Universal Robots PolyScope program: cottonMake.urp

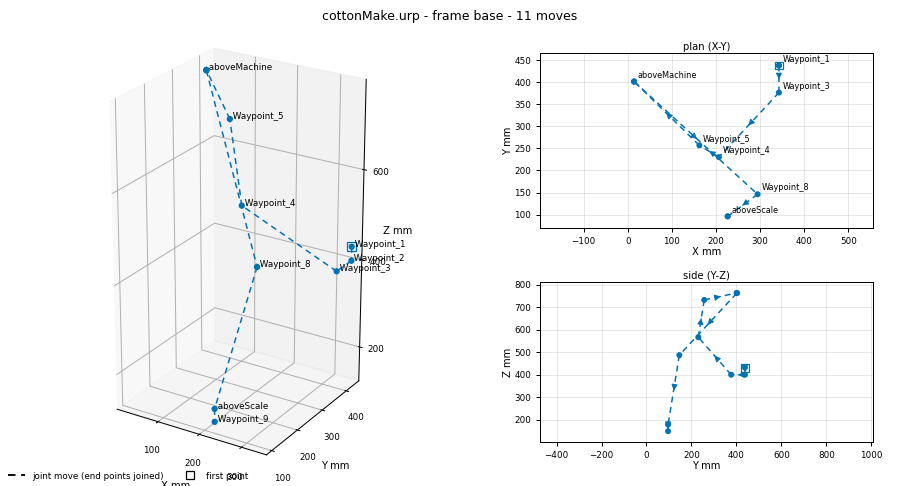
[picture p0: tool path of cottonMake.urp in frame base, 11 of 18 moves have a stored position in this frame; points joined in program order, loops and branches not executed]
Program cottonMake (installation=default directory=/programs/DavidMelin createdIn=5.12.4.1101661 lastSavedIn=5.12.4.1101661 robotSerialNumber=20225502378)
Calibrated DH parameters: a=[0.00022, -0.425328, -0.389701, 0.000059, 0.000065, 0]; d=[0.162608, 0.803456, 9.992211, -10.662202, 0.099702, 0.099559]; alpha=[1.570756, 0.001543, 0.004316, 1.570651, -1.570122, 0]; deltaTheta=[0, 0.002917, 0.116094, -0.119008, 0, -0.000001]
Robot Program (runOnlyOnce=true)
  circCenter := p[0.07107,0.64512,0.54131,0,2.2222,2.2222]
  radius := 0.12
  cBot := pose_add(circCenter, p[0,-radius,0,0,0,0])
  cLeft := pose_add(circCenter, p[-radius,0,0,0,0,0])
  cTop := pose_add(circCenter, p[0,radius,0,0,0,0])
  cRight := pose_add(circCenter, p[radius,0,0,0,0,0])
  Loops := 3
  URCap Gripper (Robotiq_Grippers, Robotiq Inc.) dataModel(position=0.0, force=0.0, speed=0.0, positionInDouble=0.0, forceInDouble=0.0, speedInDouble=0.0, slaveIds=[9], blocking=true)
  MoveJ speed 60 deg/s, acceleration 80 deg/s^2 (useActiveTCP=true) feature=Base
    Waypoint Waypoint (Variable): variable=cotonHomePos
    Waypoint Waypoint_1: TCP in base x=342.664 y=437.884 z=432.107 mm, rx=3.1413 ry=-0.0387 rz=0 rad; joints [65.941, -96.893, -90.985, -82.164, 90.259, -22.738] deg
    Waypoint Waypoint_2: TCP in base x=342.659 y=437.882 z=400.544 mm, rx=3.1413 ry=-0.0387 rz=0 rad; joints [65.938, -97.638, -94.818, -77.583, 90.259, -22.722] deg
  URCap Gripper (Robotiq_Grippers, Robotiq Inc.) dataModel(position=100.0, force=0.0, speed=0.0, positionInDouble=100.0, forceInDouble=0.0, speedInDouble=0.0, slaveIds=[9], blocking=true)
  MoveJ speed 60 deg/s, acceleration 80 deg/s^2 (useActiveTCP=true) feature=Base
    Waypoint Waypoint_3: TCP in base x=342.674 y=376.601 z=400.529 mm, rx=3.1413 ry=-0.0388 rz=0 rad; joints [62.998, -91.205, -101.8, -77.036, 90.249, -25.658] deg
    Waypoint Waypoint_4: TCP in base x=206.614 y=230.365 z=567.394 mm, rx=-2.941 ry=-0.1771 rz=0.13 rad; joints [70.752, -61.526, -101.667, -98.574, 99.079, -25.658] deg
    Waypoint Waypoint_5: TCP in base x=162.312 y=256.881 z=733.059 mm, rx=1.0793 ry=1.2981 rz=1.5955 rad; joints [107.929, -56.169, -91.557, -124.534, -6.229, -80.259] deg
    Waypoint aboveMachine: TCP in base x=14.31 y=401.62 z=764.278 mm, rx=-0.0463 ry=2.2239 rz=2.2128 rad; joints [113.283, -89.095, -46.167, -225.083, -68.031, -1.075] deg
  Loop While (checkContinuously=false) expression=Loops>0
    MoveP speed 250 mm/s, acceleration 1200 mm/s^2 (blendRadius=0.125 useActiveTCP=true) feature=Base
      Waypoint Waypoint (Variable): variable=cBot
      CircleMove (OrientationMode=UNCONSTRAINED)
        Waypoint Waypoint (Variable): variable=cRight
        Waypoint Waypoint (Variable): variable=cTop
    MoveP speed 250 mm/s, acceleration 1200 mm/s^2 (blendRadius=0.025 useActiveTCP=true) feature=Base
      Waypoint Waypoint (Variable): variable=cTop
      CircleMove (OrientationMode=UNCONSTRAINED)
        Waypoint Waypoint (Variable): variable=cLeft
        Waypoint Waypoint (Variable): variable=cBot
    Loops := Loops - 1
  MoveJ speed 60 deg/s, acceleration 80 deg/s^2 (useActiveTCP=true) feature=Base
    Waypoint aboveMachine: TCP in base x=14.31 y=401.62 z=764.278 mm, rx=-0.0463 ry=2.2239 rz=2.2128 rad; joints [113.283, -89.095, -46.167, -225.083, -68.031, -1.075] deg
    Waypoint Waypoint_6: TCP in base x=14.523 y=401.528 z=763.071 mm, rx=-1.5836 ry=0.0041 rz=0.0315 rad; joints [113.257, -89.129, -46.231, -225.448, -68.036, 181.754] deg
    Waypoint Waypoint_8: TCP in base x=294.267 y=146.163 z=487.658 mm, rx=-1.6041 ry=-0.2565 rz=0.2618 rad; joints [33.077, -80.074, -98.689, -191.144, -165.647, 171.099] deg
    Waypoint aboveScale: TCP in base x=226.497 y=96.066 z=178.622 mm, rx=-1.5818 ry=-0.3301 rz=0.3435 rad; joints [31.277, -91.949, -140.091, -142.239, -172.906, 166.771] deg
    Waypoint Waypoint_9: TCP in base x=226.483 y=96.053 z=149.343 mm, rx=-1.5818 ry=-0.3301 rz=0.3435 rad; joints [31.27, -97.11, -141.687, -135.565, -172.89, 166.689] deg
  URCap Gripper (Robotiq_Grippers, Robotiq Inc.) dataModel(position=0.0, force=0.0, speed=0.0, positionInDouble=0.0, forceInDouble=0.0, speedInDouble=0.0, slaveIds=[9], blocking=true)
